// Mitsubishi GX Works2 project: print_settings   PLC: Q02/Q02H

PROGRAM MAIN
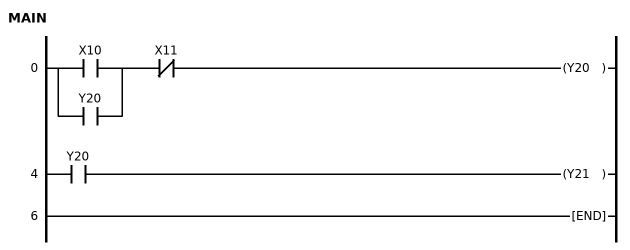
0     LD      X10
      OR      Y20
      ANI     X11
      OUT     Y20
4     LD      Y20
      OUT     Y21
6     END
END_PROGRAM
